(*
Nazwa:			FB_OEERejectionReasons
Opis:			Powód odrzuceń 
Wersja:			v0.1
Data:			2019-12-17
Autor:			DP
Urzadzenia:		
Konfiguracja:	
Info: 
- 
*)
FUNCTION_BLOCK FB_OEERejectionReason
VAR_INPUT
	bEnable: BOOL;				//Zezwolenie na pracę
	bReset:BOOL;				//Stop awaryjny nieaktywny
	udiGlobalCounter:UDINT;		//Globalny licznik
	bAddReason:BOOL;			//Dodaj pomiar
	bReason1:BOOL;
	sReason1Description:STRING;	//Nazwa stacji nr 1
	bReason2:BOOL;
	sReason2Description:STRING;	//Nazwa stacji nr 2
	bReason3:BOOL;
	sReason3Description:STRING;	//Nazwa stacji nr 3
	bReason4:BOOL;
	sReason4Description:STRING;	//Nazwa stacji nr 4
	bReason5:BOOL;
	sReason5Description:STRING;	//Nazwa stacji nr 5
	bReason6:BOOL;
	sReason6Description:STRING;	//Nazwa stacji nr 6
	bReason7:BOOL;
	sReason7Description:STRING;	//Nazwa stacji nr 7
	bReason8:BOOL;
	sReason8Description:STRING;	//Nazwa stacji nr 8
	bReason9:BOOL;
	sReason9Description:STRING;	//Nazwa stacji nr 9
	bReason10:BOOL;
	sReason10Description:STRING;	//Nazwa stacji nr 10
	bReason11:BOOL;
	sReason11Description:STRING;	//Nazwa stacji nr 11
	bReason12:BOOL;
	sReason12Description:STRING;	//Nazwa stacji nr 12
	bReason13:BOOL;
	sReason13Description:STRING;	//Nazwa stacji nr 13
	bReason14:BOOL;
	sReason14Description:STRING;	//Nazwa stacji nr 14
END_VAR

VAR_IN_OUT
	sRejectionReason			:STRING;		// Powodu odrzuceń	[symbol_odrzucenia] narazie tylko w tabeli 1
END_VAR
VAR_OUTPUT
	bDone						:BOOL;		// Powodu odrzuceń	[symbol_odrzucenia] narazie tylko w tabeli 1
END_VAR

VAR
	rtAddReason: R_TRIG;
	tonResetDone: TON;
END_VAR

ErrorHandling();
Cycle();
ManualMovements();
Statistics();

ACTION Cycle:
tonResetDone(IN:=bDone,PT:=T#300MS);
rtAddReason(CLK:=bAddReason,Q=>);
IF rtAddReason.Q THEN
	IF bReason1 THEN
		sRejectionReason:= sReason1Description;
	ELSIF bReason2 THEN		                
		sRejectionReason:= sReason2Description;
	ELSIF bReason3 THEN		                
		sRejectionReason:= sReason3Description;
	ELSIF bReason4 THEN		                
		sRejectionReason:= sReason4Description;
	ELSIF bReason5 THEN		                
		sRejectionReason:= sReason5Description;
	ELSIF bReason6 THEN		                
		sRejectionReason:= sReason6Description;
	ELSIF bReason7 THEN		                
		sRejectionReason:= sReason7Description;
	ELSIF bReason8 THEN		                
		sRejectionReason:= sReason8Description;
	ELSIF bReason9 THEN		                
		sRejectionReason:= sReason9Description;
	ELSIF bReason10 THEN		                
		sRejectionReason:= sReason10Description;
	ELSIF bReason11 THEN		                
		sRejectionReason:= sReason11Description;
	ELSIF bReason12 THEN		                
		sRejectionReason:= sReason12Description;
	ELSIF bReason13 THEN		                
		sRejectionReason:= sReason13Description;
	ELSIF bReason14 THEN		                
		sRejectionReason:= sReason14Description;

	END_IF
	bDone:= TRUE;
END_IF
IF tonResetDone.Q THEN
	bDone:= FALSE;
END_IF
END_ACTION

ACTION ErrorHandling:

END_ACTION

ACTION ManualMovements:

END_ACTION

ACTION Statistics:

END_ACTION

END_FUNCTION_BLOCK

(* stored: Version 1.1.0.1, ProductVersion 3.1.4026.13, FileIdentifier 1c109ba96410797c555c2e4be5977d79a5480cf4, FileSignature 69ebd78cc899ad70b0e1bd5fc06dc6c329653d9dd10ffccf5e718365d5999f8cb9afa9c17c0915373bc9144abbd4d03c1af7bcf3525f977828b0f59c64f2e9d487f9726b75fed238fc1b42aa66ef951f36a7e2d3c22c22e7fdf69380dd08000fa8b15aef21319f949886d3eee050050032d13aa91ab2b3a77441f14a74b318294c296140415446089f948b9b8ef420ac876349cf98fe05e12b518d5bfefcd7603dd39bafa3ddc957efc6e7bc657e60f47f532f804448041221976fe7d43f40a2d252612545128f515ab4a6446218ddfc0dcfe76bfb673d347dd3b2024edd905ec1e758b851ec017618454ed0741adfcaae002cb96ce890d3620115dd73ce1f82
   POU FB_OEERejectionReason: Id {157168b0-8e99-4670-b737-cd1e6e3754e6}, SpecialFunc None
   Action Cycle: Id {bef05546-ae52-47ef-8bf9-6551b8fcf721}
   Action ErrorHandling: Id {d16e4274-a31a-4b46-b749-440766d76761}
   Action ManualMovements: Id {f84853de-bcc0-4499-bedb-656d6c9b400e}
   Action Statistics: Id {4d7bdb75-d901-4776-b8f6-2c1089062138} *)
